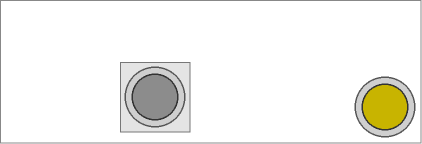
VISUALIZATION Visualization  // 422x144
    Lamp1 (350,72 70x70), variable: GVL_1.Blinke_Lampe, style: Lamp-Lamp1-Yellow
    PushSwitch (120,62 70x70), variable: GVL_1.Viso_Schalter, behaviour: TOGGLE, style: Switch-PushSwitch-Gray
END_VISUALIZATION

(* stored: Version 1.1.0.1, ProductVersion 3.1.4022.9
   Visu Visualization: Id {d33fe873-4efe-4f45-9ad3-64e91749d57a} *)
